{attribute 'analysis' := '-33'}
PROGRAM INTERNAL PRG_UnitTests
VAR
{IF defined (UNIT_TEST)}

{END_IF}
END_VAR

{IF defined (UNIT_TEST)}
PRG_ParsingPrimitiveTests();
PRG_RoundTripTests();
PRG_WritingPrimitiveTests();
PRG_MessageTests();
PRG_WireFormatTests();
PRG_EnumTests();
PRG_RepeatedFieldTests();
PRG_HelperTests();
PRG_SpanTests();
PRG_IssuesTests();
TcUnit.RUN();

{END_IF}

END_PROGRAM

(* stored: Version 1.1.0.1
   POU PRG_UnitTests: Id {c62e4430-fc3d-4856-ad8a-4ac6f6b51a31}, SpecialFunc None *)
